{attribute 'qualified_only'}
{attribute 'strict'}
{attribute 'to_string'}
TYPE E_MachineState :
(
    PowerUp      := 0,
    Fault        := 1,
    Stopping     := 2,
    Stopped      := 3,
    Initialising := 4,
    ReadyToStart := 5,
    AutoCycle    := 6,
    Manual       := 7
);
END_TYPE

(* stored: Version 1.1.0.1, ProductVersion 3.1.4026.18
   DUT E_MachineState: Id {473e1156-2b87-40d4-a57b-c37602246c60} *)
